TYPE aocHmiCommands_TypeStruct :
STRUCT
	
	aocExecute : BOOL;

END_STRUCT
END_TYPE

(* stored: Version 1.1.0.1
   DUT aocHmiCommands_TypeStruct: Id {0c8830b3-4dcf-4aba-97ee-3eb5f91e0d6b} *)
